{attribute 'qualified_only'}
VAR_GLOBAL
	// Meldeleuchte "Schliessen"
	P1: BOOL;
	// Motor LL (Öffnen)
	Q1: BOOL;
	// Motor RL (Schliessen)
	Q2: BOOL;
END_VAR

(* stored: Version 1.1.0.1, ProductVersion 3.1.4024.5
   GVL SimDA: Id {efa3d63a-96e1-4204-b1e7-9f3703bd4f03} *)
